// TIA Portal V19 export
DATA_BLOCK "next2DB"   // DB333
{ S7_Optimized_Access := 'TRUE' }
// stored: AutoNumber false, MemoryReserve 100
BEGIN
END_DATA_BLOCK
